// TIA Portal project "SS1_Tom" (V19)

(* hardware
DEVICE "SIMATIC 1200 station_1"  S71200.Device
   slot 0: "S7-1200 rack"  Rack  V1.0
   slot 1: "PLC_1"  CPU 1214C DC/DC/DC  6ES7 214-1AG40-0XB0  V4.0
   slot 3: "AQ1 x 12 bits_1"  6ES7 232-4HA30-0XB0  V1.0
*)

// ===== PLC "PLC_1"  CPU 1214C DC/DC/DC =====

VAR_GLOBAL   // PLC tag table "Default tag table"
   "STOP" AT %I0.1 : Bool;   // Pushbutton Momentary N.C.
   "START" AT %I0.0 : Bool;   // Pushbutton Momentary N.O.
   "PL1_OFF" AT %Q0.0 : Bool;   // Pilot Light 1 OFF (RED)
   "PL2_ON" AT %Q0.1 : Bool;   // Pilot Light 1 ON (Green)
   "MOTOR" AT %Q0.2 : Bool;   // Motor Control
END_VAR

ORGANIZATION_BLOCK "Main"   // OB1, SCL, ProgramCycle
TITLE = "Main Program Sweep (Cycle)"
{ S7_Optimized_Access := 'TRUE' }
VERSION : 0.1
BEGIN
   //START-STOP pushbuttons to turn On MOTOR
   "MOTOR":="STOP"AND ("START"OR"MOTOR");


   //Indicators status based on MOTOR On or Off
   "PL1_OFF" := NOT "MOTOR";
   "PL2_ON" := "MOTOR";
END_ORGANIZATION_BLOCK